// TIA Portal V20 export
TYPE "LBP_typeNCVariableToken"
TITLE = LBP_ReadVar and LBP_WriteVar Input Interface / Interface d'entrée LBP_ReadVar et LBP_WriteVar
// User Data Type for LBP_ReadVar[FB2] and LBP_WriteVar[FB3] Input Parameter Addrx / Type de données utilisateur pour les paramètres d'entrée Addrx LBP_ReadVar[FB2] et LBP_WriteVar[FB3]
   STRUCT
      syntaxId : Byte;   // syntax ID / ID de syntaxe
      areaAndUnit : Byte;   // area and unit / zone et unité
      column : Word;   // column / colonne
      row : Word;   // row / ligne
      blockType : Byte;   // block type / type de bloc
      numberOfRows : Byte;   // number of rows / nombre de lignes
      dataTypeCode : Byte;   // data type code / code de type de données
      length : Byte;   // length of data type / longueur de type de données
   END_STRUCT;
END_TYPE
